// TIA Portal V17 export
// export: Created 2025-03-07T09:18:06.0998876Z, ExportSetting WithDefaults, DisplayName Totally Integrated Automation Portal, DisplayVersion V17 Update 8, DisplayName TIA Portal Openness, DisplayVersion V17 Update 8, DisplayName TIA Portal Version Control Interface, DisplayVersion V17, DisplayName SINAMICS Startdrive Advanced, DisplayVersion V17 SP2, DisplayName SINAMICS Startdrive G110M, G120, G120C, G120D, G120P, G115D, DisplayVersion V17 SP2, DisplayName SINAMICS Startdrive G130, G150, S120, S150, SINAMICS MV, S210, DisplayVersion V17 SP2, DisplayName STEP 7 Professional, DisplayVersion V17 Update 8, DisplayName SINUMERIK ONE STEP 7 Toolbox, DisplayVersion V17 Update 12, DisplayName SINUMERIK 840D sl STEP 7 Toolbox, DisplayVersion V17 Update 12, DisplayName STEP 7 Safety, DisplayVersion V17 Update 6, DisplayName WinCC Advanced, DisplayVersion V17 Update 8
FUNCTION "FC1285_UNIT_02_STATION_3_MASTER_MEASUREMENT" : Void   // FC1285, LAD
{ S7_Optimized_Access := 'FALSE' }
AUTHOR : ETXETAR
VERSION : 1.0
// stored: AutoNumber false, IsIECCheckEnabled false, SetENOAutomatically false, UDAEnableTagReadback false
   VAR CONSTANT
      FC_NUMBER : DInt := 1285;
   END_VAR
   VAR_TEMP   // added for the SCL form of the ladder/FBD networks
      _w1 : Bool;
      _w2 : Bool;
   END_VAR
BEGIN

REGION Network 1: GENERAL CONDITIONS
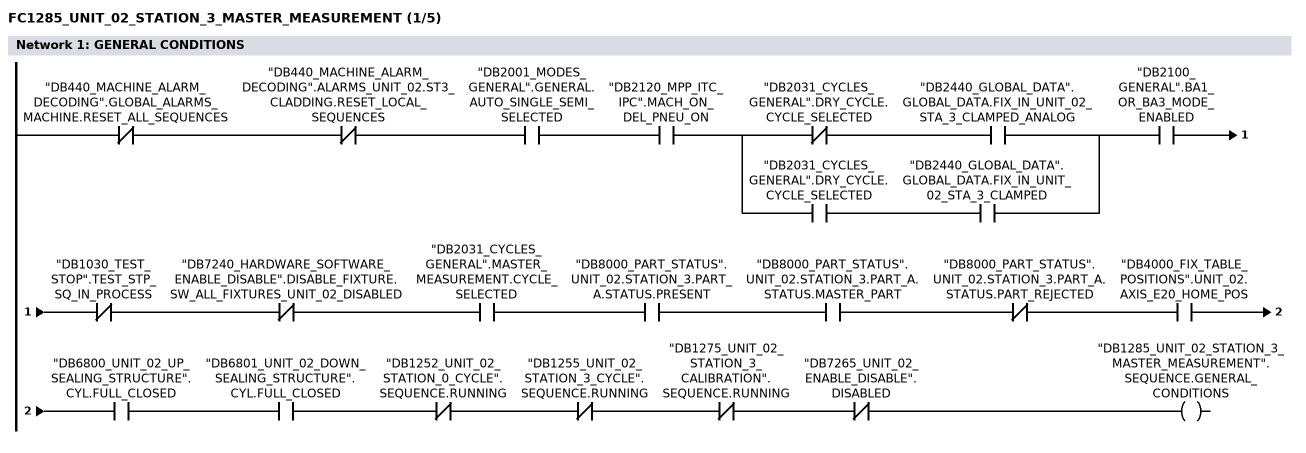
   RUNG wire#powerrail
      I_Contact( "DB440_MACHINE_ALARM_DECODING".GLOBAL_ALARMS_MACHINE.RESET_ALL_SEQUENCES )
      I_Contact( "DB440_MACHINE_ALARM_DECODING".ALARMS_UNIT_02.ST3_CLADDING.RESET_LOCAL_SEQUENCES )
      Contact( "DB2001_MODES_GENERAL".GENERAL.AUTO_SINGLE_SEMI_SELECTED )
      Contact( "DB2120_MPP_ITC_IPC".MACH_ON_DEL_PNEU_ON )
      wire#w1
      I_Contact( "DB2031_CYCLES_GENERAL".DRY_CYCLE.CYCLE_SELECTED )
      Contact( "DB2440_GLOBAL_DATA".GLOBAL_DATA.FIX_IN_UNIT_02_STA_3_CLAMPED_ANALOG )
      wire#w2
      Contact( "DB2100_GENERAL".BA1_OR_BA3_MODE_ENABLED )
      I_Contact( "DB1030_TEST_STOP".TEST_STP_SQ_IN_PROCESS )
      I_Contact( "DB7240_HARDWARE_SOFTWARE_ENABLE_DISABLE".DISABLE_FIXTURE.SW_ALL_FIXTURES_UNIT_02_DISABLED )
      Contact( "DB2031_CYCLES_GENERAL".MASTER_MEASUREMENT.CYCLE_SELECTED )
      Contact( "DB8000_PART_STATUS".UNIT_02.STATION_3.PART_A.STATUS.PRESENT )
      Contact( "DB8000_PART_STATUS".UNIT_02.STATION_3.PART_A.STATUS.MASTER_PART )
      I_Contact( "DB8000_PART_STATUS".UNIT_02.STATION_3.PART_A.STATUS.PART_REJECTED )
      Contact( "DB4000_FIX_TABLE_POSITIONS".UNIT_02.AXIS_E20_HOME_POS )
      Contact( "DB6800_UNIT_02_UP_SEALING_STRUCTURE".CYL.FULL_CLOSED )
      Contact( "DB6801_UNIT_02_DOWN_SEALING_STRUCTURE".CYL.FULL_CLOSED )
      I_Contact( "DB1252_UNIT_02_STATION_0_CYCLE".SEQUENCE.RUNNING )
      I_Contact( "DB1255_UNIT_02_STATION_3_CYCLE".SEQUENCE.RUNNING )
      I_Contact( "DB1275_UNIT_02_STATION_3_CALIBRATION".SEQUENCE.RUNNING )
      I_Contact( "DB7265_UNIT_02_ENABLE_DISABLE".DISABLED )
      Coil( "DB1285_UNIT_02_STATION_3_MASTER_MEASUREMENT".SEQUENCE.GENERAL_CONDITIONS )
   END_RUNG
   RUNG wire#w1
      Contact( "DB2031_CYCLES_GENERAL".DRY_CYCLE.CYCLE_SELECTED )
      Contact( "DB2440_GLOBAL_DATA".GLOBAL_DATA.FIX_IN_UNIT_02_STA_3_CLAMPED )
   END_RUNG wire#w2
   // the same network as SCL:
   "DB1285_UNIT_02_STATION_3_MASTER_MEASUREMENT".SEQUENCE.GENERAL_CONDITIONS := NOT "DB440_MACHINE_ALARM_DECODING".GLOBAL_ALARMS_MACHINE.RESET_ALL_SEQUENCES AND NOT "DB440_MACHINE_ALARM_DECODING".ALARMS_UNIT_02.ST3_CLADDING.RESET_LOCAL_SEQUENCES AND "DB2001_MODES_GENERAL".GENERAL.AUTO_SINGLE_SEMI_SELECTED AND "DB2120_MPP_ITC_IPC".MACH_ON_DEL_PNEU_ON AND ((NOT "DB2031_CYCLES_GENERAL".DRY_CYCLE.CYCLE_SELECTED AND "DB2440_GLOBAL_DATA".GLOBAL_DATA.FIX_IN_UNIT_02_STA_3_CLAMPED_ANALOG) OR ("DB2031_CYCLES_GENERAL".DRY_CYCLE.CYCLE_SELECTED AND "DB2440_GLOBAL_DATA".GLOBAL_DATA.FIX_IN_UNIT_02_STA_3_CLAMPED)) AND "DB2100_GENERAL".BA1_OR_BA3_MODE_ENABLED AND NOT "DB1030_TEST_STOP".TEST_STP_SQ_IN_PROCESS AND NOT "DB7240_HARDWARE_SOFTWARE_ENABLE_DISABLE".DISABLE_FIXTURE.SW_ALL_FIXTURES_UNIT_02_DISABLED AND "DB2031_CYCLES_GENERAL".MASTER_MEASUREMENT.CYCLE_SELECTED AND "DB8000_PART_STATUS".UNIT_02.STATION_3.PART_A.STATUS.PRESENT AND "DB8000_PART_STATUS".UNIT_02.STATION_3.PART_A.STATUS.MASTER_PART AND NOT "DB8000_PART_STATUS".UNIT_02.STATION_3.PART_A.STATUS.PART_REJECTED AND "DB4000_FIX_TABLE_POSITIONS".UNIT_02.AXIS_E20_HOME_POS AND "DB6800_UNIT_02_UP_SEALING_STRUCTURE".CYL.FULL_CLOSED AND "DB6801_UNIT_02_DOWN_SEALING_STRUCTURE".CYL.FULL_CLOSED AND NOT "DB1252_UNIT_02_STATION_0_CYCLE".SEQUENCE.RUNNING AND NOT "DB1255_UNIT_02_STATION_3_CYCLE".SEQUENCE.RUNNING AND NOT "DB1275_UNIT_02_STATION_3_CALIBRATION".SEQUENCE.RUNNING AND NOT "DB7265_UNIT_02_ENABLE_DISABLE".DISABLED;
END_REGION

REGION Network 2: OPERATOR HELP
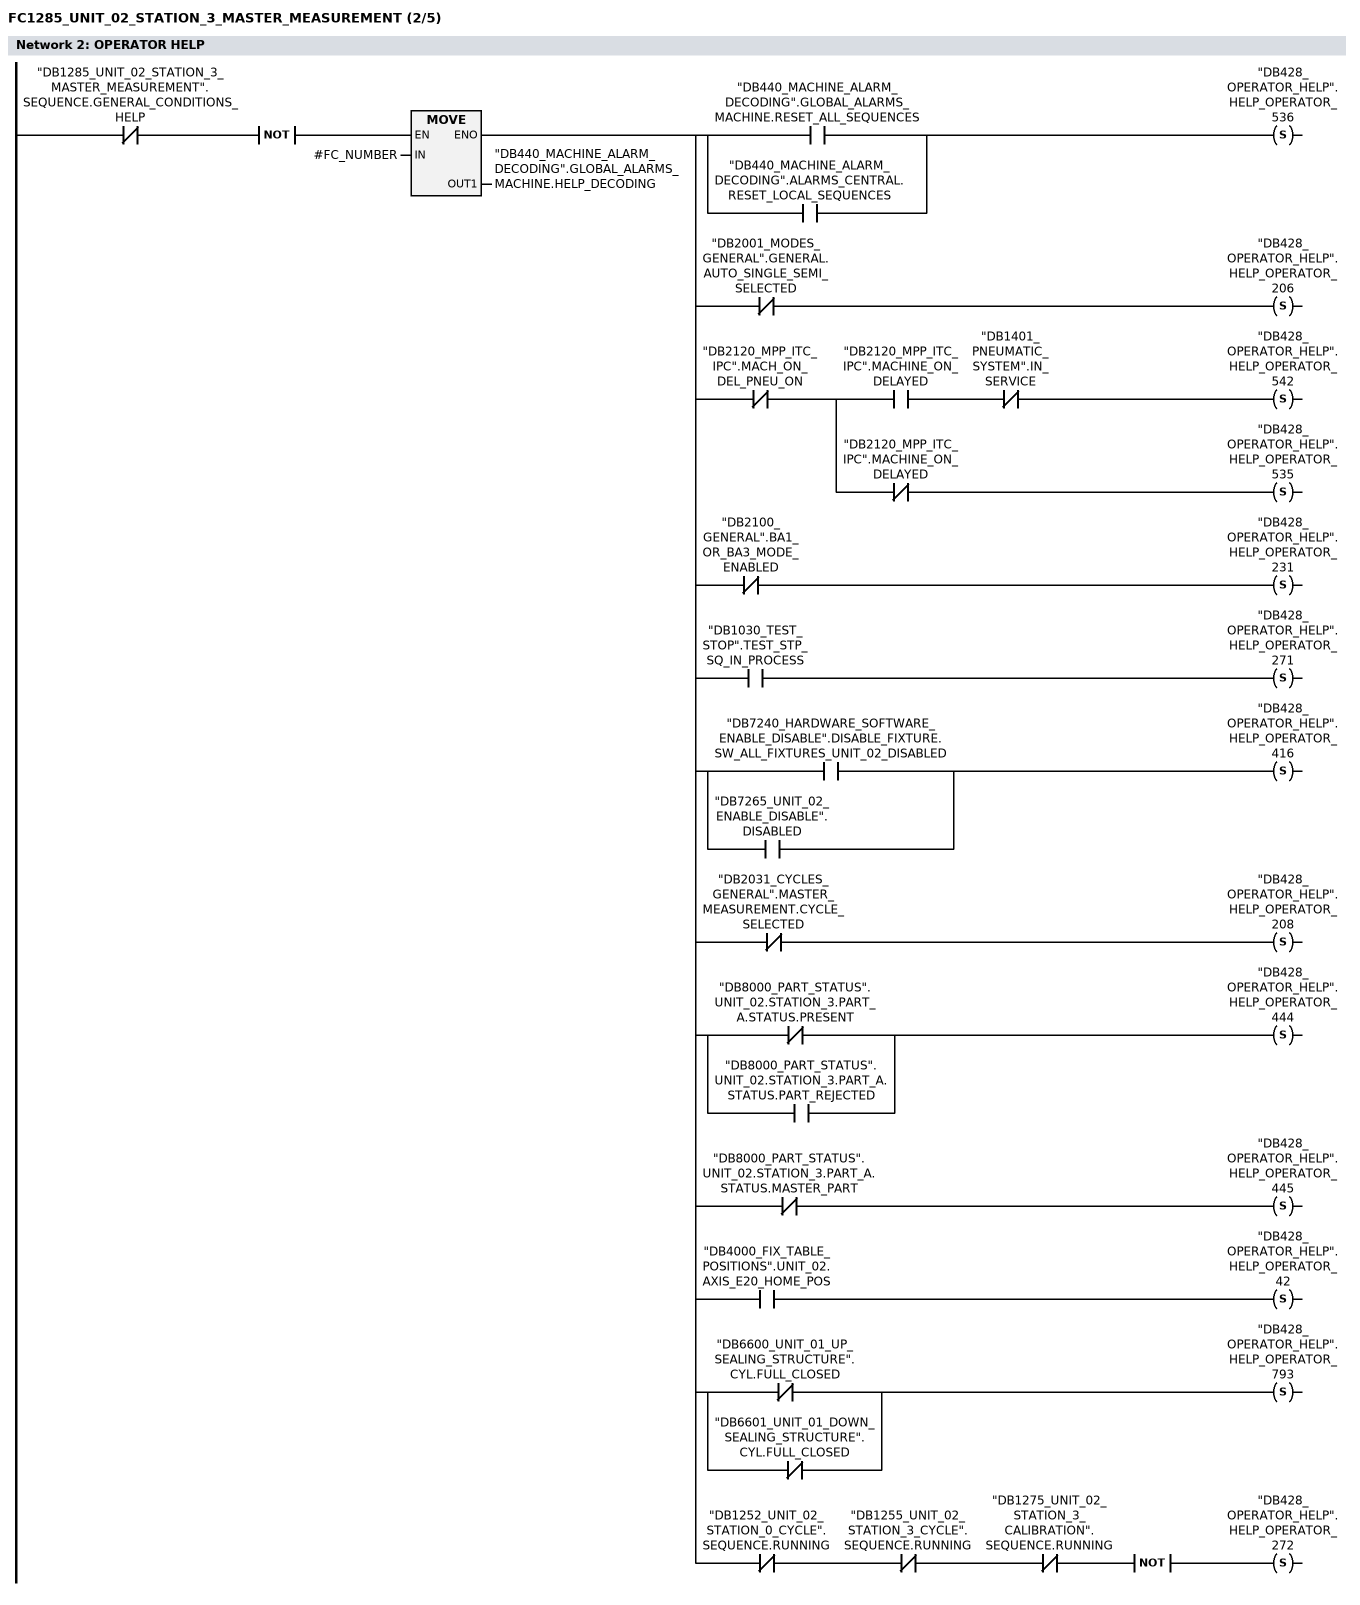
   RUNG wire#powerrail
      I_Contact( "DB1285_UNIT_02_STATION_3_MASTER_MEASUREMENT".SEQUENCE.GENERAL_CONDITIONS_HELP )
      Not()
      { S7_GenerateENO := "TRUE" } Move(in := #FC_NUMBER, out1 => "DB440_MACHINE_ALARM_DECODING".GLOBAL_ALARMS_MACHINE.HELP_DECODING)
      wire#w1
      Contact( "DB440_MACHINE_ALARM_DECODING".GLOBAL_ALARMS_MACHINE.RESET_ALL_SEQUENCES )
      wire#w2
      S_Coil( "DB428_OPERATOR_HELP".HELP_OPERATOR_536 )
   END_RUNG
   RUNG wire#w1
      Contact( "DB440_MACHINE_ALARM_DECODING".ALARMS_CENTRAL.RESET_LOCAL_SEQUENCES )
   END_RUNG wire#w2
   RUNG wire#w1
      I_Contact( "DB2001_MODES_GENERAL".GENERAL.AUTO_SINGLE_SEMI_SELECTED )
      S_Coil( "DB428_OPERATOR_HELP".HELP_OPERATOR_206 )
   END_RUNG
   RUNG wire#w1
      I_Contact( "DB2120_MPP_ITC_IPC".MACH_ON_DEL_PNEU_ON )
      wire#w3
      Contact( "DB2120_MPP_ITC_IPC".MACHINE_ON_DELAYED )
      I_Contact( "DB1401_PNEUMATIC_SYSTEM".IN_SERVICE )
      S_Coil( "DB428_OPERATOR_HELP".HELP_OPERATOR_542 )
   END_RUNG
   RUNG wire#w3
      I_Contact( "DB2120_MPP_ITC_IPC".MACHINE_ON_DELAYED )
      S_Coil( "DB428_OPERATOR_HELP".HELP_OPERATOR_535 )
   END_RUNG
   RUNG wire#w1
      I_Contact( "DB2100_GENERAL".BA1_OR_BA3_MODE_ENABLED )
      S_Coil( "DB428_OPERATOR_HELP".HELP_OPERATOR_231 )
   END_RUNG
   RUNG wire#w1
      Contact( "DB1030_TEST_STOP".TEST_STP_SQ_IN_PROCESS )
      S_Coil( "DB428_OPERATOR_HELP".HELP_OPERATOR_271 )
   END_RUNG
   RUNG wire#w1
      Contact( "DB7240_HARDWARE_SOFTWARE_ENABLE_DISABLE".DISABLE_FIXTURE.SW_ALL_FIXTURES_UNIT_02_DISABLED )
      wire#w4
      S_Coil( "DB428_OPERATOR_HELP".HELP_OPERATOR_416 )
   END_RUNG
   RUNG wire#w1
      Contact( "DB7265_UNIT_02_ENABLE_DISABLE".DISABLED )
   END_RUNG wire#w4
   RUNG wire#w1
      I_Contact( "DB2031_CYCLES_GENERAL".MASTER_MEASUREMENT.CYCLE_SELECTED )
      S_Coil( "DB428_OPERATOR_HELP".HELP_OPERATOR_208 )
   END_RUNG
   RUNG wire#w1
      I_Contact( "DB8000_PART_STATUS".UNIT_02.STATION_3.PART_A.STATUS.PRESENT )
      wire#w5
      S_Coil( "DB428_OPERATOR_HELP".HELP_OPERATOR_444 )
   END_RUNG
   RUNG wire#w1
      Contact( "DB8000_PART_STATUS".UNIT_02.STATION_3.PART_A.STATUS.PART_REJECTED )
   END_RUNG wire#w5
   RUNG wire#w1
      I_Contact( "DB8000_PART_STATUS".UNIT_02.STATION_3.PART_A.STATUS.MASTER_PART )
      S_Coil( "DB428_OPERATOR_HELP".HELP_OPERATOR_445 )
   END_RUNG
   RUNG wire#w1
      Contact( "DB4000_FIX_TABLE_POSITIONS".UNIT_02.AXIS_E20_HOME_POS )
      S_Coil( "DB428_OPERATOR_HELP".HELP_OPERATOR_42 )
   END_RUNG
   RUNG wire#w1
      I_Contact( "DB6600_UNIT_01_UP_SEALING_STRUCTURE".CYL.FULL_CLOSED )
      wire#w6
      S_Coil( "DB428_OPERATOR_HELP".HELP_OPERATOR_793 )
   END_RUNG
   RUNG wire#w1
      I_Contact( "DB6601_UNIT_01_DOWN_SEALING_STRUCTURE".CYL.FULL_CLOSED )
   END_RUNG wire#w6
   RUNG wire#w1
      I_Contact( "DB1252_UNIT_02_STATION_0_CYCLE".SEQUENCE.RUNNING )
      I_Contact( "DB1255_UNIT_02_STATION_3_CYCLE".SEQUENCE.RUNNING )
      I_Contact( "DB1275_UNIT_02_STATION_3_CALIBRATION".SEQUENCE.RUNNING )
      Not()
      S_Coil( "DB428_OPERATOR_HELP".HELP_OPERATOR_272 )
   END_RUNG
   // the same network as SCL:
   // ENO of a box is taken as its EN; it also drops when the box reports an error
   #_w1 := NOT (NOT "DB1285_UNIT_02_STATION_3_MASTER_MEASUREMENT".SEQUENCE.GENERAL_CONDITIONS_HELP);
   IF #_w1 THEN "DB440_MACHINE_ALARM_DECODING".GLOBAL_ALARMS_MACHINE.HELP_DECODING := #FC_NUMBER; END_IF;
   IF #_w1 AND ("DB440_MACHINE_ALARM_DECODING".GLOBAL_ALARMS_MACHINE.RESET_ALL_SEQUENCES OR "DB440_MACHINE_ALARM_DECODING".ALARMS_CENTRAL.RESET_LOCAL_SEQUENCES) THEN
       "DB428_OPERATOR_HELP".HELP_OPERATOR_536 := TRUE;
   END_IF;
   IF #_w1 AND NOT "DB2001_MODES_GENERAL".GENERAL.AUTO_SINGLE_SEMI_SELECTED THEN
       "DB428_OPERATOR_HELP".HELP_OPERATOR_206 := TRUE;
   END_IF;
   #_w2 := #_w1 AND NOT "DB2120_MPP_ITC_IPC".MACH_ON_DEL_PNEU_ON;
   IF #_w2 AND "DB2120_MPP_ITC_IPC".MACHINE_ON_DELAYED AND NOT "DB1401_PNEUMATIC_SYSTEM".IN_SERVICE THEN
       "DB428_OPERATOR_HELP".HELP_OPERATOR_542 := TRUE;
   END_IF;
   IF #_w2 AND NOT "DB2120_MPP_ITC_IPC".MACHINE_ON_DELAYED THEN
       "DB428_OPERATOR_HELP".HELP_OPERATOR_535 := TRUE;
   END_IF;
   IF #_w1 AND NOT "DB2100_GENERAL".BA1_OR_BA3_MODE_ENABLED THEN
       "DB428_OPERATOR_HELP".HELP_OPERATOR_231 := TRUE;
   END_IF;
   IF #_w1 AND "DB1030_TEST_STOP".TEST_STP_SQ_IN_PROCESS THEN
       "DB428_OPERATOR_HELP".HELP_OPERATOR_271 := TRUE;
   END_IF;
   IF #_w1 AND ("DB7240_HARDWARE_SOFTWARE_ENABLE_DISABLE".DISABLE_FIXTURE.SW_ALL_FIXTURES_UNIT_02_DISABLED OR "DB7265_UNIT_02_ENABLE_DISABLE".DISABLED) THEN
       "DB428_OPERATOR_HELP".HELP_OPERATOR_416 := TRUE;
   END_IF;
   IF #_w1 AND NOT "DB2031_CYCLES_GENERAL".MASTER_MEASUREMENT.CYCLE_SELECTED THEN
       "DB428_OPERATOR_HELP".HELP_OPERATOR_208 := TRUE;
   END_IF;
   IF #_w1 AND (NOT "DB8000_PART_STATUS".UNIT_02.STATION_3.PART_A.STATUS.PRESENT OR "DB8000_PART_STATUS".UNIT_02.STATION_3.PART_A.STATUS.PART_REJECTED) THEN
       "DB428_OPERATOR_HELP".HELP_OPERATOR_444 := TRUE;
   END_IF;
   IF #_w1 AND NOT "DB8000_PART_STATUS".UNIT_02.STATION_3.PART_A.STATUS.MASTER_PART THEN
       "DB428_OPERATOR_HELP".HELP_OPERATOR_445 := TRUE;
   END_IF;
   IF #_w1 AND "DB4000_FIX_TABLE_POSITIONS".UNIT_02.AXIS_E20_HOME_POS THEN
       "DB428_OPERATOR_HELP".HELP_OPERATOR_42 := TRUE;
   END_IF;
   IF #_w1 AND (NOT "DB6600_UNIT_01_UP_SEALING_STRUCTURE".CYL.FULL_CLOSED OR NOT "DB6601_UNIT_01_DOWN_SEALING_STRUCTURE".CYL.FULL_CLOSED) THEN
       "DB428_OPERATOR_HELP".HELP_OPERATOR_793 := TRUE;
   END_IF;
   IF NOT (#_w1 AND NOT "DB1252_UNIT_02_STATION_0_CYCLE".SEQUENCE.RUNNING AND NOT "DB1255_UNIT_02_STATION_3_CYCLE".SEQUENCE.RUNNING AND NOT "DB1275_UNIT_02_STATION_3_CALIBRATION".SEQUENCE.RUNNING) THEN
       "DB428_OPERATOR_HELP".HELP_OPERATOR_272 := TRUE;
   END_IF;
END_REGION

REGION Network 3: INITIAL CONDITIONS
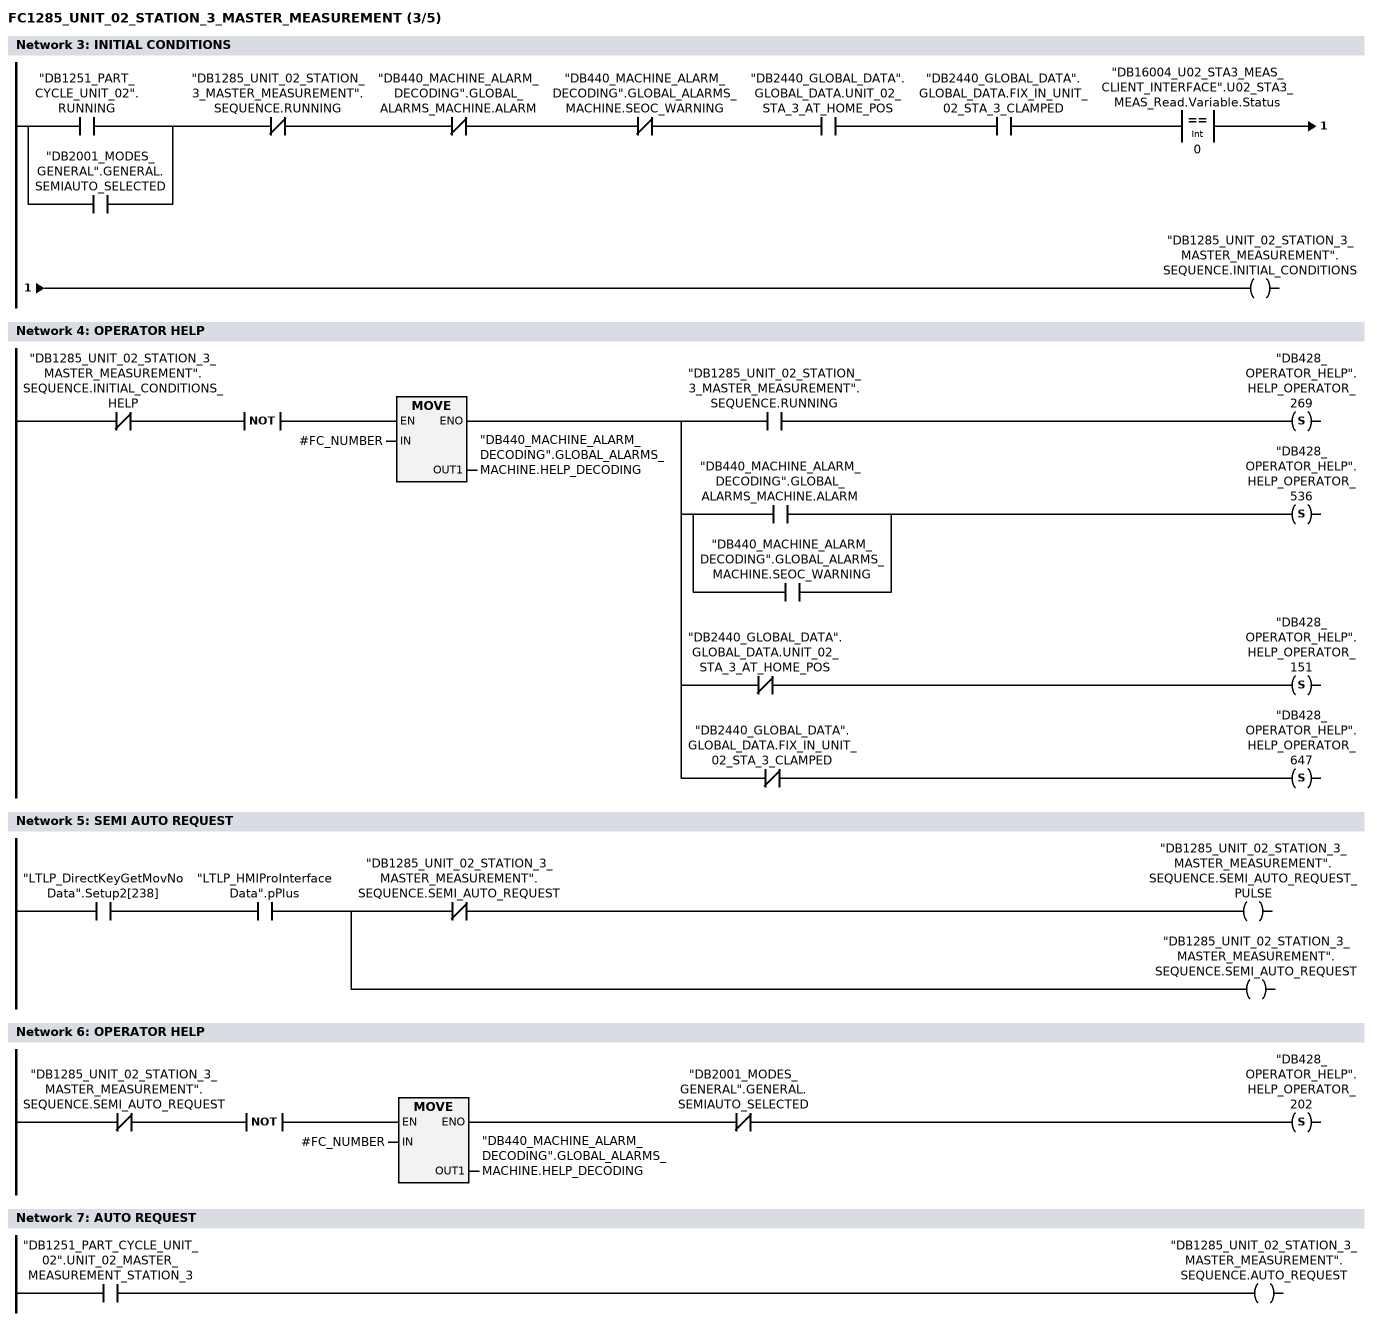
   RUNG wire#powerrail
      Contact( "DB1251_PART_CYCLE_UNIT_02".RUNNING )
      wire#w1
      I_Contact( "DB1285_UNIT_02_STATION_3_MASTER_MEASUREMENT".SEQUENCE.RUNNING )
      I_Contact( "DB440_MACHINE_ALARM_DECODING".GLOBAL_ALARMS_MACHINE.ALARM )
      I_Contact( "DB440_MACHINE_ALARM_DECODING".GLOBAL_ALARMS_MACHINE.SEOC_WARNING )
      Contact( "DB2440_GLOBAL_DATA".GLOBAL_DATA.UNIT_02_STA_3_AT_HOME_POS )
      Contact( "DB2440_GLOBAL_DATA".GLOBAL_DATA.FIX_IN_UNIT_02_STA_3_CLAMPED )
      { S7_Templates := "SrcType := Int" } EQ_Contact(in1 := "DB16004_U02_STA3_MEAS_CLIENT_INTERFACE".U02_STA3_MEAS_Read.Variable.Status, in2 := 0)
      Coil( "DB1285_UNIT_02_STATION_3_MASTER_MEASUREMENT".SEQUENCE.INITIAL_CONDITIONS )
   END_RUNG
   RUNG wire#powerrail
      Contact( "DB2001_MODES_GENERAL".GENERAL.SEMIAUTO_SELECTED )
   END_RUNG wire#w1
   // the same network as SCL:
   "DB1285_UNIT_02_STATION_3_MASTER_MEASUREMENT".SEQUENCE.INITIAL_CONDITIONS := ("DB1251_PART_CYCLE_UNIT_02".RUNNING OR "DB2001_MODES_GENERAL".GENERAL.SEMIAUTO_SELECTED) AND NOT "DB1285_UNIT_02_STATION_3_MASTER_MEASUREMENT".SEQUENCE.RUNNING AND NOT "DB440_MACHINE_ALARM_DECODING".GLOBAL_ALARMS_MACHINE.ALARM AND NOT "DB440_MACHINE_ALARM_DECODING".GLOBAL_ALARMS_MACHINE.SEOC_WARNING AND "DB2440_GLOBAL_DATA".GLOBAL_DATA.UNIT_02_STA_3_AT_HOME_POS AND "DB2440_GLOBAL_DATA".GLOBAL_DATA.FIX_IN_UNIT_02_STA_3_CLAMPED AND ("DB16004_U02_STA3_MEAS_CLIENT_INTERFACE".U02_STA3_MEAS_Read.Variable.Status = 0);
END_REGION

REGION Network 4: OPERATOR HELP
   RUNG wire#powerrail
      I_Contact( "DB1285_UNIT_02_STATION_3_MASTER_MEASUREMENT".SEQUENCE.INITIAL_CONDITIONS_HELP )
      Not()
      { S7_GenerateENO := "TRUE" } Move(in := #FC_NUMBER, out1 => "DB440_MACHINE_ALARM_DECODING".GLOBAL_ALARMS_MACHINE.HELP_DECODING)
      wire#w1
      Contact( "DB1285_UNIT_02_STATION_3_MASTER_MEASUREMENT".SEQUENCE.RUNNING )
      S_Coil( "DB428_OPERATOR_HELP".HELP_OPERATOR_269 )
   END_RUNG
   RUNG wire#w1
      Contact( "DB440_MACHINE_ALARM_DECODING".GLOBAL_ALARMS_MACHINE.ALARM )
      wire#w2
      S_Coil( "DB428_OPERATOR_HELP".HELP_OPERATOR_536 )
   END_RUNG
   RUNG wire#w1
      Contact( "DB440_MACHINE_ALARM_DECODING".GLOBAL_ALARMS_MACHINE.SEOC_WARNING )
   END_RUNG wire#w2
   RUNG wire#w1
      I_Contact( "DB2440_GLOBAL_DATA".GLOBAL_DATA.UNIT_02_STA_3_AT_HOME_POS )
      S_Coil( "DB428_OPERATOR_HELP".HELP_OPERATOR_151 )
   END_RUNG
   RUNG wire#w1
      I_Contact( "DB2440_GLOBAL_DATA".GLOBAL_DATA.FIX_IN_UNIT_02_STA_3_CLAMPED )
      S_Coil( "DB428_OPERATOR_HELP".HELP_OPERATOR_647 )
   END_RUNG
   // the same network as SCL:
   // ENO of a box is taken as its EN; it also drops when the box reports an error
   #_w1 := NOT (NOT "DB1285_UNIT_02_STATION_3_MASTER_MEASUREMENT".SEQUENCE.INITIAL_CONDITIONS_HELP);
   IF #_w1 THEN "DB440_MACHINE_ALARM_DECODING".GLOBAL_ALARMS_MACHINE.HELP_DECODING := #FC_NUMBER; END_IF;
   IF #_w1 AND "DB1285_UNIT_02_STATION_3_MASTER_MEASUREMENT".SEQUENCE.RUNNING THEN
       "DB428_OPERATOR_HELP".HELP_OPERATOR_269 := TRUE;
   END_IF;
   IF #_w1 AND ("DB440_MACHINE_ALARM_DECODING".GLOBAL_ALARMS_MACHINE.ALARM OR "DB440_MACHINE_ALARM_DECODING".GLOBAL_ALARMS_MACHINE.SEOC_WARNING) THEN
       "DB428_OPERATOR_HELP".HELP_OPERATOR_536 := TRUE;
   END_IF;
   IF #_w1 AND NOT "DB2440_GLOBAL_DATA".GLOBAL_DATA.UNIT_02_STA_3_AT_HOME_POS THEN
       "DB428_OPERATOR_HELP".HELP_OPERATOR_151 := TRUE;
   END_IF;
   IF #_w1 AND NOT "DB2440_GLOBAL_DATA".GLOBAL_DATA.FIX_IN_UNIT_02_STA_3_CLAMPED THEN
       "DB428_OPERATOR_HELP".HELP_OPERATOR_647 := TRUE;
   END_IF;
END_REGION

REGION Network 5: SEMI AUTO REQUEST
   RUNG wire#powerrail
      Contact( "LTLP_DirectKeyGetMovNoData".Setup2[238] )
      Contact( "LTLP_HMIProInterfaceData".pPlus )
      wire#w1
      I_Contact( "DB1285_UNIT_02_STATION_3_MASTER_MEASUREMENT".SEQUENCE.SEMI_AUTO_REQUEST )
      Coil( "DB1285_UNIT_02_STATION_3_MASTER_MEASUREMENT".SEQUENCE.SEMI_AUTO_REQUEST_PULSE )
   END_RUNG
   RUNG wire#w1
      Coil( "DB1285_UNIT_02_STATION_3_MASTER_MEASUREMENT".SEQUENCE.SEMI_AUTO_REQUEST )
   END_RUNG
   // the same network as SCL:
   #_w1 := "LTLP_DirectKeyGetMovNoData".Setup2[238] AND "LTLP_HMIProInterfaceData".pPlus;
   "DB1285_UNIT_02_STATION_3_MASTER_MEASUREMENT".SEQUENCE.SEMI_AUTO_REQUEST_PULSE := #_w1 AND NOT "DB1285_UNIT_02_STATION_3_MASTER_MEASUREMENT".SEQUENCE.SEMI_AUTO_REQUEST;
   "DB1285_UNIT_02_STATION_3_MASTER_MEASUREMENT".SEQUENCE.SEMI_AUTO_REQUEST := #_w1;
END_REGION

REGION Network 6: OPERATOR HELP
   RUNG wire#powerrail
      I_Contact( "DB1285_UNIT_02_STATION_3_MASTER_MEASUREMENT".SEQUENCE.SEMI_AUTO_REQUEST )
      Not()
      { S7_GenerateENO := "TRUE" } Move(in := #FC_NUMBER, out1 => "DB440_MACHINE_ALARM_DECODING".GLOBAL_ALARMS_MACHINE.HELP_DECODING)
      I_Contact( "DB2001_MODES_GENERAL".GENERAL.SEMIAUTO_SELECTED )
      S_Coil( "DB428_OPERATOR_HELP".HELP_OPERATOR_202 )
   END_RUNG
   // the same network as SCL:
   // ENO of a box is taken as its EN; it also drops when the box reports an error
   #_w1 := NOT (NOT "DB1285_UNIT_02_STATION_3_MASTER_MEASUREMENT".SEQUENCE.SEMI_AUTO_REQUEST);
   IF #_w1 THEN "DB440_MACHINE_ALARM_DECODING".GLOBAL_ALARMS_MACHINE.HELP_DECODING := #FC_NUMBER; END_IF;
   IF #_w1 AND NOT "DB2001_MODES_GENERAL".GENERAL.SEMIAUTO_SELECTED THEN
       "DB428_OPERATOR_HELP".HELP_OPERATOR_202 := TRUE;
   END_IF;
END_REGION

REGION Network 7: AUTO REQUEST
   RUNG wire#powerrail
      Contact( "DB1251_PART_CYCLE_UNIT_02".UNIT_02_MASTER_MEASUREMENT_STATION_3 )
      Coil( "DB1285_UNIT_02_STATION_3_MASTER_MEASUREMENT".SEQUENCE.AUTO_REQUEST )
   END_RUNG
   // the same network as SCL:
   "DB1285_UNIT_02_STATION_3_MASTER_MEASUREMENT".SEQUENCE.AUTO_REQUEST := "DB1251_PART_CYCLE_UNIT_02".UNIT_02_MASTER_MEASUREMENT_STATION_3;
END_REGION

REGION Network 8: REQUEST
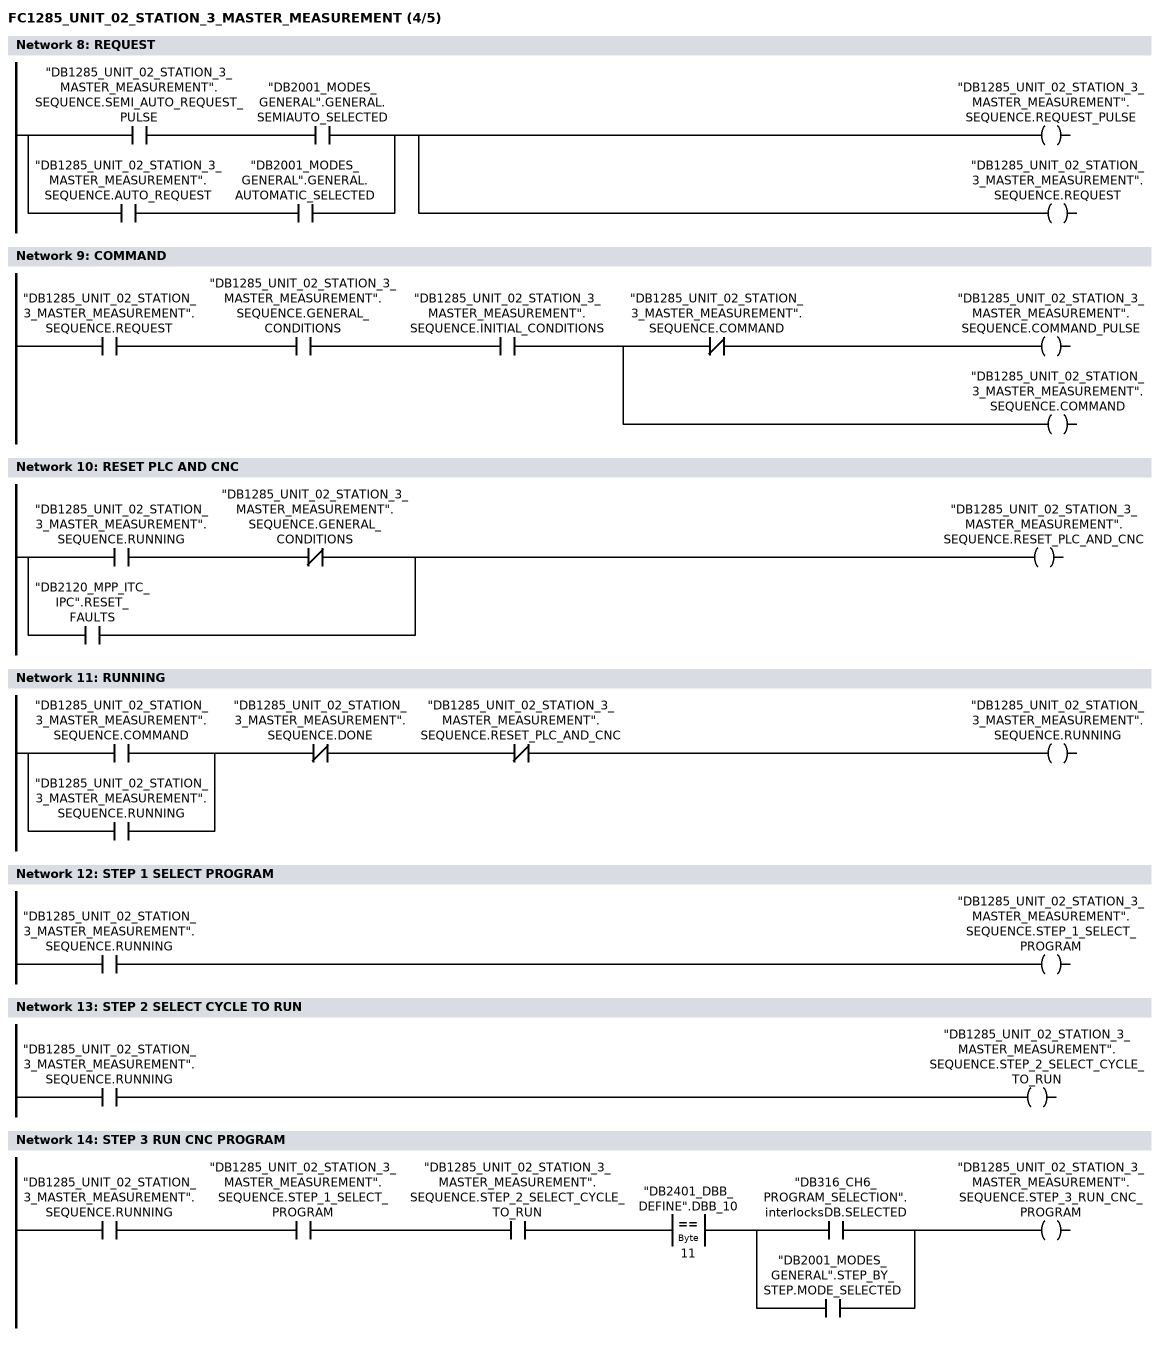
   RUNG wire#powerrail
      Contact( "DB1285_UNIT_02_STATION_3_MASTER_MEASUREMENT".SEQUENCE.SEMI_AUTO_REQUEST_PULSE )
      Contact( "DB2001_MODES_GENERAL".GENERAL.SEMIAUTO_SELECTED )
      wire#w1
      Coil( "DB1285_UNIT_02_STATION_3_MASTER_MEASUREMENT".SEQUENCE.REQUEST_PULSE )
   END_RUNG
   RUNG wire#powerrail
      Contact( "DB1285_UNIT_02_STATION_3_MASTER_MEASUREMENT".SEQUENCE.AUTO_REQUEST )
      Contact( "DB2001_MODES_GENERAL".GENERAL.AUTOMATIC_SELECTED )
   END_RUNG wire#w1
   RUNG wire#w1
      Coil( "DB1285_UNIT_02_STATION_3_MASTER_MEASUREMENT".SEQUENCE.REQUEST )
   END_RUNG
   // the same network as SCL:
   "DB1285_UNIT_02_STATION_3_MASTER_MEASUREMENT".SEQUENCE.REQUEST_PULSE := ("DB1285_UNIT_02_STATION_3_MASTER_MEASUREMENT".SEQUENCE.SEMI_AUTO_REQUEST_PULSE AND "DB2001_MODES_GENERAL".GENERAL.SEMIAUTO_SELECTED) OR ("DB1285_UNIT_02_STATION_3_MASTER_MEASUREMENT".SEQUENCE.AUTO_REQUEST AND "DB2001_MODES_GENERAL".GENERAL.AUTOMATIC_SELECTED);
   "DB1285_UNIT_02_STATION_3_MASTER_MEASUREMENT".SEQUENCE.REQUEST := "DB1285_UNIT_02_STATION_3_MASTER_MEASUREMENT".SEQUENCE.REQUEST_PULSE;
END_REGION

REGION Network 9: COMMAND
   RUNG wire#powerrail
      Contact( "DB1285_UNIT_02_STATION_3_MASTER_MEASUREMENT".SEQUENCE.REQUEST )
      Contact( "DB1285_UNIT_02_STATION_3_MASTER_MEASUREMENT".SEQUENCE.GENERAL_CONDITIONS )
      Contact( "DB1285_UNIT_02_STATION_3_MASTER_MEASUREMENT".SEQUENCE.INITIAL_CONDITIONS )
      wire#w1
      I_Contact( "DB1285_UNIT_02_STATION_3_MASTER_MEASUREMENT".SEQUENCE.COMMAND )
      Coil( "DB1285_UNIT_02_STATION_3_MASTER_MEASUREMENT".SEQUENCE.COMMAND_PULSE )
   END_RUNG
   RUNG wire#w1
      Coil( "DB1285_UNIT_02_STATION_3_MASTER_MEASUREMENT".SEQUENCE.COMMAND )
   END_RUNG
   // the same network as SCL:
   #_w1 := "DB1285_UNIT_02_STATION_3_MASTER_MEASUREMENT".SEQUENCE.REQUEST AND "DB1285_UNIT_02_STATION_3_MASTER_MEASUREMENT".SEQUENCE.GENERAL_CONDITIONS AND "DB1285_UNIT_02_STATION_3_MASTER_MEASUREMENT".SEQUENCE.INITIAL_CONDITIONS;
   "DB1285_UNIT_02_STATION_3_MASTER_MEASUREMENT".SEQUENCE.COMMAND_PULSE := #_w1 AND NOT "DB1285_UNIT_02_STATION_3_MASTER_MEASUREMENT".SEQUENCE.COMMAND;
   "DB1285_UNIT_02_STATION_3_MASTER_MEASUREMENT".SEQUENCE.COMMAND := #_w1;
END_REGION

REGION Network 10: RESET PLC AND CNC
   RUNG wire#powerrail
      Contact( "DB1285_UNIT_02_STATION_3_MASTER_MEASUREMENT".SEQUENCE.RUNNING )
      I_Contact( "DB1285_UNIT_02_STATION_3_MASTER_MEASUREMENT".SEQUENCE.GENERAL_CONDITIONS )
      wire#w1
      Coil( "DB1285_UNIT_02_STATION_3_MASTER_MEASUREMENT".SEQUENCE.RESET_PLC_AND_CNC )
   END_RUNG
   RUNG wire#powerrail
      Contact( "DB2120_MPP_ITC_IPC".RESET_FAULTS )
   END_RUNG wire#w1
   // the same network as SCL:
   "DB1285_UNIT_02_STATION_3_MASTER_MEASUREMENT".SEQUENCE.RESET_PLC_AND_CNC := ("DB1285_UNIT_02_STATION_3_MASTER_MEASUREMENT".SEQUENCE.RUNNING AND NOT "DB1285_UNIT_02_STATION_3_MASTER_MEASUREMENT".SEQUENCE.GENERAL_CONDITIONS) OR "DB2120_MPP_ITC_IPC".RESET_FAULTS;
END_REGION

REGION Network 11: RUNNING
   RUNG wire#powerrail
      Contact( "DB1285_UNIT_02_STATION_3_MASTER_MEASUREMENT".SEQUENCE.COMMAND )
      wire#w1
      I_Contact( "DB1285_UNIT_02_STATION_3_MASTER_MEASUREMENT".SEQUENCE.DONE )
      I_Contact( "DB1285_UNIT_02_STATION_3_MASTER_MEASUREMENT".SEQUENCE.RESET_PLC_AND_CNC )
      Coil( "DB1285_UNIT_02_STATION_3_MASTER_MEASUREMENT".SEQUENCE.RUNNING )
   END_RUNG
   RUNG wire#powerrail
      Contact( "DB1285_UNIT_02_STATION_3_MASTER_MEASUREMENT".SEQUENCE.RUNNING )
   END_RUNG wire#w1
   // the same network as SCL:
   "DB1285_UNIT_02_STATION_3_MASTER_MEASUREMENT".SEQUENCE.RUNNING := ("DB1285_UNIT_02_STATION_3_MASTER_MEASUREMENT".SEQUENCE.COMMAND OR "DB1285_UNIT_02_STATION_3_MASTER_MEASUREMENT".SEQUENCE.RUNNING) AND NOT "DB1285_UNIT_02_STATION_3_MASTER_MEASUREMENT".SEQUENCE.DONE AND NOT "DB1285_UNIT_02_STATION_3_MASTER_MEASUREMENT".SEQUENCE.RESET_PLC_AND_CNC;
END_REGION

REGION Network 12: STEP 1 SELECT PROGRAM
   RUNG wire#powerrail
      Contact( "DB1285_UNIT_02_STATION_3_MASTER_MEASUREMENT".SEQUENCE.RUNNING )
      Coil( "DB1285_UNIT_02_STATION_3_MASTER_MEASUREMENT".SEQUENCE.STEP_1_SELECT_PROGRAM )
   END_RUNG
   // the same network as SCL:
   "DB1285_UNIT_02_STATION_3_MASTER_MEASUREMENT".SEQUENCE.STEP_1_SELECT_PROGRAM := "DB1285_UNIT_02_STATION_3_MASTER_MEASUREMENT".SEQUENCE.RUNNING;
END_REGION

REGION Network 13: STEP 2 SELECT CYCLE TO RUN
   RUNG wire#powerrail
      Contact( "DB1285_UNIT_02_STATION_3_MASTER_MEASUREMENT".SEQUENCE.RUNNING )
      Coil( "DB1285_UNIT_02_STATION_3_MASTER_MEASUREMENT".SEQUENCE.STEP_2_SELECT_CYCLE_TO_RUN )
   END_RUNG
   // the same network as SCL:
   "DB1285_UNIT_02_STATION_3_MASTER_MEASUREMENT".SEQUENCE.STEP_2_SELECT_CYCLE_TO_RUN := "DB1285_UNIT_02_STATION_3_MASTER_MEASUREMENT".SEQUENCE.RUNNING;
END_REGION

REGION Network 14: STEP 3 RUN CNC PROGRAM
   RUNG wire#powerrail
      Contact( "DB1285_UNIT_02_STATION_3_MASTER_MEASUREMENT".SEQUENCE.RUNNING )
      Contact( "DB1285_UNIT_02_STATION_3_MASTER_MEASUREMENT".SEQUENCE.STEP_1_SELECT_PROGRAM )
      Contact( "DB1285_UNIT_02_STATION_3_MASTER_MEASUREMENT".SEQUENCE.STEP_2_SELECT_CYCLE_TO_RUN )
      { S7_Templates := "SrcType := Byte" } EQ_Contact(in1 := "DB2401_DBB_DEFINE".DBB_10, in2 := 11)
      wire#w1
      Contact( "DB316_CH6_PROGRAM_SELECTION".interlocksDB.SELECTED )
      wire#w2
      Coil( "DB1285_UNIT_02_STATION_3_MASTER_MEASUREMENT".SEQUENCE.STEP_3_RUN_CNC_PROGRAM )
   END_RUNG
   RUNG wire#w1
      Contact( "DB2001_MODES_GENERAL".STEP_BY_STEP.MODE_SELECTED )
   END_RUNG wire#w2
   // the same network as SCL:
   "DB1285_UNIT_02_STATION_3_MASTER_MEASUREMENT".SEQUENCE.STEP_3_RUN_CNC_PROGRAM := "DB1285_UNIT_02_STATION_3_MASTER_MEASUREMENT".SEQUENCE.RUNNING AND "DB1285_UNIT_02_STATION_3_MASTER_MEASUREMENT".SEQUENCE.STEP_1_SELECT_PROGRAM AND "DB1285_UNIT_02_STATION_3_MASTER_MEASUREMENT".SEQUENCE.STEP_2_SELECT_CYCLE_TO_RUN AND ("DB2401_DBB_DEFINE".DBB_10 = 11) AND ("DB316_CH6_PROGRAM_SELECTION".interlocksDB.SELECTED OR "DB2001_MODES_GENERAL".STEP_BY_STEP.MODE_SELECTED);
END_REGION

REGION Network 15: DONE
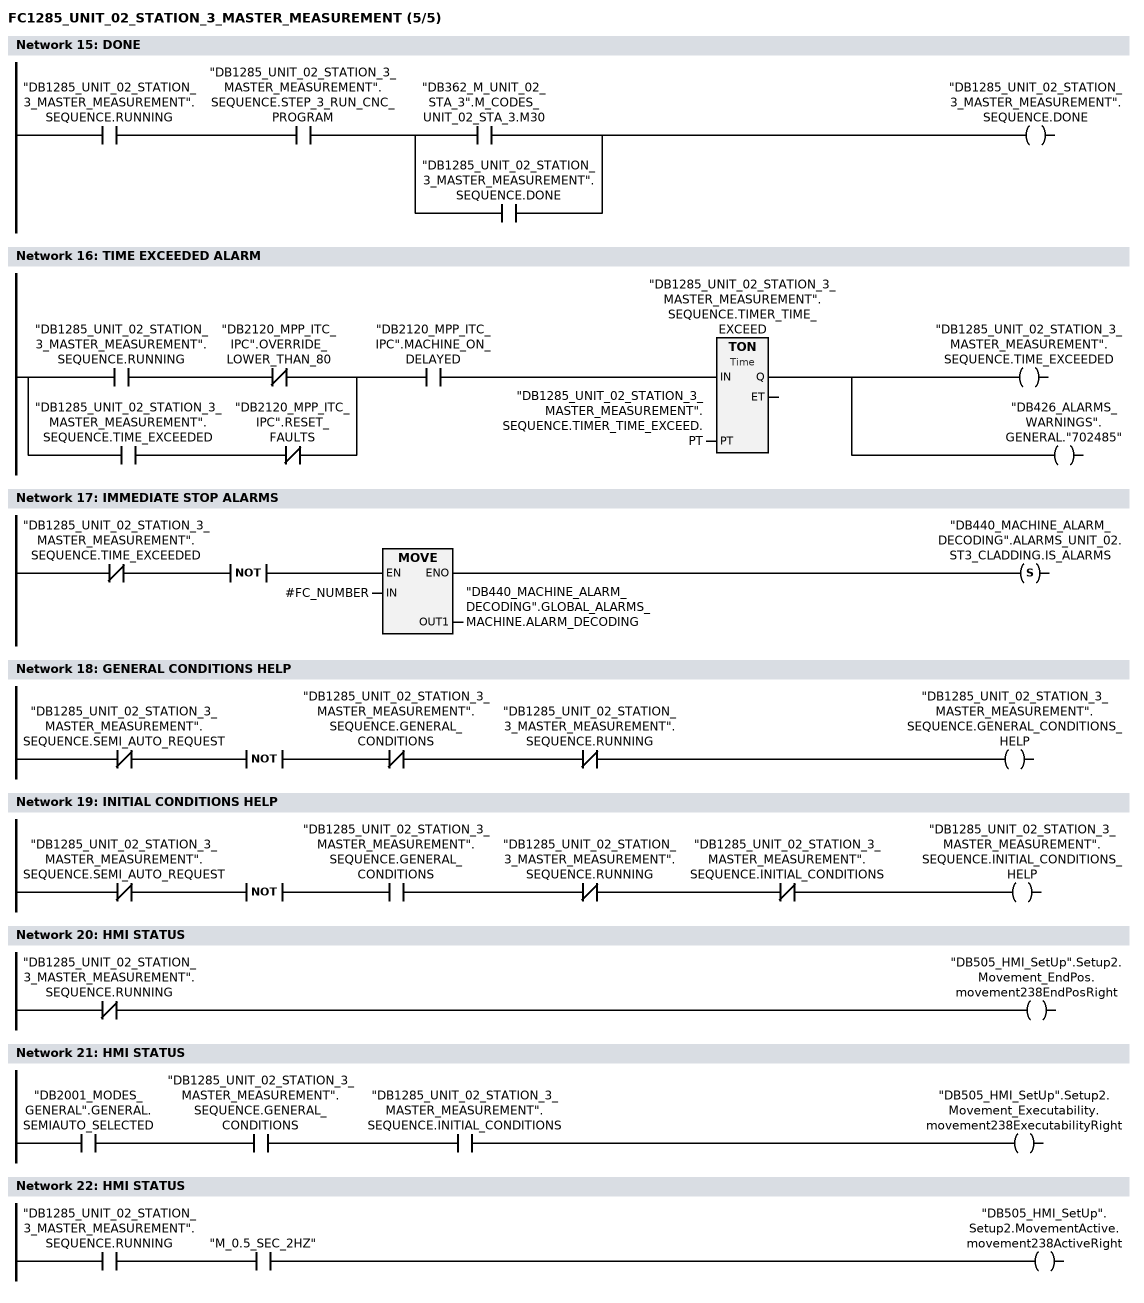
   RUNG wire#powerrail
      Contact( "DB1285_UNIT_02_STATION_3_MASTER_MEASUREMENT".SEQUENCE.RUNNING )
      Contact( "DB1285_UNIT_02_STATION_3_MASTER_MEASUREMENT".SEQUENCE.STEP_3_RUN_CNC_PROGRAM )
      wire#w1
      Contact( "DB362_M_UNIT_02_STA_3".M_CODES_UNIT_02_STA_3.M30 )
      wire#w2
      Coil( "DB1285_UNIT_02_STATION_3_MASTER_MEASUREMENT".SEQUENCE.DONE )
   END_RUNG
   RUNG wire#w1
      Contact( "DB1285_UNIT_02_STATION_3_MASTER_MEASUREMENT".SEQUENCE.DONE )
   END_RUNG wire#w2
   // the same network as SCL:
   "DB1285_UNIT_02_STATION_3_MASTER_MEASUREMENT".SEQUENCE.DONE := "DB1285_UNIT_02_STATION_3_MASTER_MEASUREMENT".SEQUENCE.RUNNING AND "DB1285_UNIT_02_STATION_3_MASTER_MEASUREMENT".SEQUENCE.STEP_3_RUN_CNC_PROGRAM AND ("DB362_M_UNIT_02_STA_3".M_CODES_UNIT_02_STA_3.M30 OR "DB1285_UNIT_02_STATION_3_MASTER_MEASUREMENT".SEQUENCE.DONE);
END_REGION

REGION Network 16: TIME EXCEEDED ALARM
   RUNG wire#powerrail
      Contact( "DB1285_UNIT_02_STATION_3_MASTER_MEASUREMENT".SEQUENCE.RUNNING )
      I_Contact( "DB2120_MPP_ITC_IPC".OVERRIDE_LOWER_THAN_80 )
      wire#w1
      Contact( "DB2120_MPP_ITC_IPC".MACHINE_ON_DELAYED )
      { S7_Templates := "time_type := Time" } "DB1285_UNIT_02_STATION_3_MASTER_MEASUREMENT".SEQUENCE.TIMER_TIME_EXCEED.TON(pt := "DB1285_UNIT_02_STATION_3_MASTER_MEASUREMENT".SEQUENCE.TIMER_TIME_EXCEED.PT, et =>)
      wire#w2
      Coil( "DB1285_UNIT_02_STATION_3_MASTER_MEASUREMENT".SEQUENCE.TIME_EXCEEDED )
   END_RUNG
   RUNG wire#powerrail
      Contact( "DB1285_UNIT_02_STATION_3_MASTER_MEASUREMENT".SEQUENCE.TIME_EXCEEDED )
      I_Contact( "DB2120_MPP_ITC_IPC".RESET_FAULTS )
   END_RUNG wire#w1
   RUNG wire#w2
      Coil( "DB426_ALARMS_WARNINGS".GENERAL."702485" )
   END_RUNG
   // the same network as SCL:
   "DB1285_UNIT_02_STATION_3_MASTER_MEASUREMENT".SEQUENCE.TIMER_TIME_EXCEED.TON(IN := (("DB1285_UNIT_02_STATION_3_MASTER_MEASUREMENT".SEQUENCE.RUNNING AND NOT "DB2120_MPP_ITC_IPC".OVERRIDE_LOWER_THAN_80) OR ("DB1285_UNIT_02_STATION_3_MASTER_MEASUREMENT".SEQUENCE.TIME_EXCEEDED AND NOT "DB2120_MPP_ITC_IPC".RESET_FAULTS)) AND "DB2120_MPP_ITC_IPC".MACHINE_ON_DELAYED,
                           PT := "DB1285_UNIT_02_STATION_3_MASTER_MEASUREMENT".SEQUENCE.TIMER_TIME_EXCEED.PT);
   "DB1285_UNIT_02_STATION_3_MASTER_MEASUREMENT".SEQUENCE.TIME_EXCEEDED := "DB1285_UNIT_02_STATION_3_MASTER_MEASUREMENT".SEQUENCE.TIMER_TIME_EXCEED.Q;
   "DB426_ALARMS_WARNINGS".GENERAL."702485" := "DB1285_UNIT_02_STATION_3_MASTER_MEASUREMENT".SEQUENCE.TIMER_TIME_EXCEED.Q;
END_REGION

REGION Network 17: IMMEDIATE STOP ALARMS
   RUNG wire#powerrail
      I_Contact( "DB1285_UNIT_02_STATION_3_MASTER_MEASUREMENT".SEQUENCE.TIME_EXCEEDED )
      Not()
      { S7_GenerateENO := "TRUE" } Move(in := #FC_NUMBER, out1 => "DB440_MACHINE_ALARM_DECODING".GLOBAL_ALARMS_MACHINE.ALARM_DECODING)
      S_Coil( "DB440_MACHINE_ALARM_DECODING".ALARMS_UNIT_02.ST3_CLADDING.IS_ALARMS )
   END_RUNG
   // the same network as SCL:
   // ENO of a box is taken as its EN; it also drops when the box reports an error
   IF NOT (NOT "DB1285_UNIT_02_STATION_3_MASTER_MEASUREMENT".SEQUENCE.TIME_EXCEEDED) THEN
       "DB440_MACHINE_ALARM_DECODING".GLOBAL_ALARMS_MACHINE.ALARM_DECODING := #FC_NUMBER;
       "DB440_MACHINE_ALARM_DECODING".ALARMS_UNIT_02.ST3_CLADDING.IS_ALARMS := TRUE;
   END_IF;
END_REGION

REGION Network 18: GENERAL CONDITIONS HELP
   RUNG wire#powerrail
      I_Contact( "DB1285_UNIT_02_STATION_3_MASTER_MEASUREMENT".SEQUENCE.SEMI_AUTO_REQUEST )
      Not()
      I_Contact( "DB1285_UNIT_02_STATION_3_MASTER_MEASUREMENT".SEQUENCE.GENERAL_CONDITIONS )
      I_Contact( "DB1285_UNIT_02_STATION_3_MASTER_MEASUREMENT".SEQUENCE.RUNNING )
      Coil( "DB1285_UNIT_02_STATION_3_MASTER_MEASUREMENT".SEQUENCE.GENERAL_CONDITIONS_HELP )
   END_RUNG
   // the same network as SCL:
   "DB1285_UNIT_02_STATION_3_MASTER_MEASUREMENT".SEQUENCE.GENERAL_CONDITIONS_HELP := NOT (NOT "DB1285_UNIT_02_STATION_3_MASTER_MEASUREMENT".SEQUENCE.SEMI_AUTO_REQUEST) AND NOT "DB1285_UNIT_02_STATION_3_MASTER_MEASUREMENT".SEQUENCE.GENERAL_CONDITIONS AND NOT "DB1285_UNIT_02_STATION_3_MASTER_MEASUREMENT".SEQUENCE.RUNNING;
END_REGION

REGION Network 19: INITIAL CONDITIONS HELP
   RUNG wire#powerrail
      I_Contact( "DB1285_UNIT_02_STATION_3_MASTER_MEASUREMENT".SEQUENCE.SEMI_AUTO_REQUEST )
      Not()
      Contact( "DB1285_UNIT_02_STATION_3_MASTER_MEASUREMENT".SEQUENCE.GENERAL_CONDITIONS )
      I_Contact( "DB1285_UNIT_02_STATION_3_MASTER_MEASUREMENT".SEQUENCE.RUNNING )
      I_Contact( "DB1285_UNIT_02_STATION_3_MASTER_MEASUREMENT".SEQUENCE.INITIAL_CONDITIONS )
      Coil( "DB1285_UNIT_02_STATION_3_MASTER_MEASUREMENT".SEQUENCE.INITIAL_CONDITIONS_HELP )
   END_RUNG
   // the same network as SCL:
   "DB1285_UNIT_02_STATION_3_MASTER_MEASUREMENT".SEQUENCE.INITIAL_CONDITIONS_HELP := NOT (NOT "DB1285_UNIT_02_STATION_3_MASTER_MEASUREMENT".SEQUENCE.SEMI_AUTO_REQUEST) AND "DB1285_UNIT_02_STATION_3_MASTER_MEASUREMENT".SEQUENCE.GENERAL_CONDITIONS AND NOT "DB1285_UNIT_02_STATION_3_MASTER_MEASUREMENT".SEQUENCE.RUNNING AND NOT "DB1285_UNIT_02_STATION_3_MASTER_MEASUREMENT".SEQUENCE.INITIAL_CONDITIONS;
END_REGION

REGION Network 20: HMI STATUS
   RUNG wire#powerrail
      I_Contact( "DB1285_UNIT_02_STATION_3_MASTER_MEASUREMENT".SEQUENCE.RUNNING )
      Coil( "DB505_HMI_SetUp".Setup2.Movement_EndPos.movement238EndPosRight )
   END_RUNG
   // the same network as SCL:
   "DB505_HMI_SetUp".Setup2.Movement_EndPos.movement238EndPosRight := NOT "DB1285_UNIT_02_STATION_3_MASTER_MEASUREMENT".SEQUENCE.RUNNING;
END_REGION

REGION Network 21: HMI STATUS
   RUNG wire#powerrail
      Contact( "DB2001_MODES_GENERAL".GENERAL.SEMIAUTO_SELECTED )
      Contact( "DB1285_UNIT_02_STATION_3_MASTER_MEASUREMENT".SEQUENCE.GENERAL_CONDITIONS )
      Contact( "DB1285_UNIT_02_STATION_3_MASTER_MEASUREMENT".SEQUENCE.INITIAL_CONDITIONS )
      Coil( "DB505_HMI_SetUp".Setup2.Movement_Executability.movement238ExecutabilityRight )
   END_RUNG
   // the same network as SCL:
   "DB505_HMI_SetUp".Setup2.Movement_Executability.movement238ExecutabilityRight := "DB2001_MODES_GENERAL".GENERAL.SEMIAUTO_SELECTED AND "DB1285_UNIT_02_STATION_3_MASTER_MEASUREMENT".SEQUENCE.GENERAL_CONDITIONS AND "DB1285_UNIT_02_STATION_3_MASTER_MEASUREMENT".SEQUENCE.INITIAL_CONDITIONS;
END_REGION

REGION Network 22: HMI STATUS
   RUNG wire#powerrail
      Contact( "DB1285_UNIT_02_STATION_3_MASTER_MEASUREMENT".SEQUENCE.RUNNING )
      Contact( "M_0.5_SEC_2HZ" )
      Coil( "DB505_HMI_SetUp".Setup2.MovementActive.movement238ActiveRight )
   END_RUNG
   // the same network as SCL:
   "DB505_HMI_SetUp".Setup2.MovementActive.movement238ActiveRight := "DB1285_UNIT_02_STATION_3_MASTER_MEASUREMENT".SEQUENCE.RUNNING AND "M_0.5_SEC_2HZ";
END_REGION
END_FUNCTION
